ABB RobotStudio station: proyectoRueda.rspag

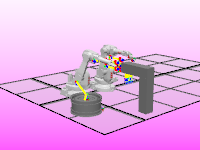
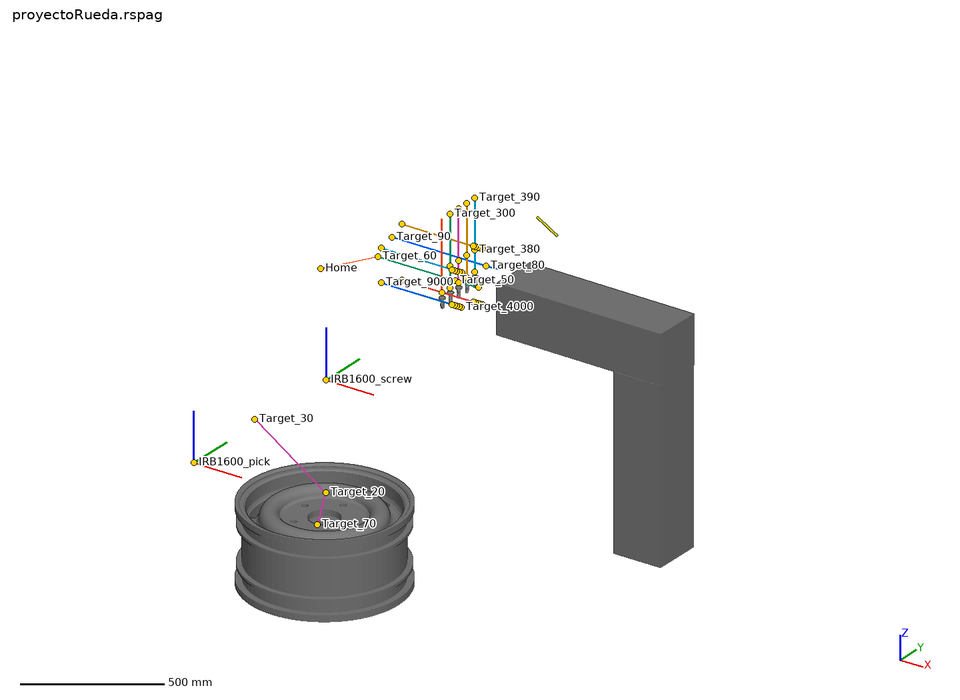
[picture v1: parts stored in the station drawn from their meshes, with robot base, taught points and paths (robot models come from the ABB library and are not in the file)]
--- station ---
Station Versión2 (saved by RobotStudio 21.2.9526.0)
Controller Controlador3, task T_ROB1: task frame (RAPID world) sits at (0, 800, 0) mm in the station
Controller Controlador1
  mechanical unit ROB_1: IRB1600_pick, 6 joints, base frame (0, 0, 0) mm
Controller Controlador3
  mechanical unit ROB_1: IRB1600_screw, 6 joints, base frame (0, 0, 0) mm
Layout (positions relative to the parent item):
  - Pieza_8 [part] at (1800, 250, 0) mm, size 200 x 200 x 700 mm
  - base_rueda [part] at (1800, 450, 700) mm, rotated rx 0 ry 0 rz -0.44 deg, size 700 x 200 x 200 mm
  - IRB1600_pick [mechanism, from Robots\IRB1600_6_120_G_02.rslib] at (0, 0, 0) mm; joint values [0.4149, 0.36, -0.1352, -2.0394, 0.4688, 2.0869] (rad or m)
  - Mi_Ventosa [smart component, from Downloads\1217c23c-7d3e-48fb-b7d3-d1b2005a3c2bMi_Ventosa.rslib] at (890.68, 363.73, 797.26) mm, rotated rx 0 ry 90 rz 0 deg
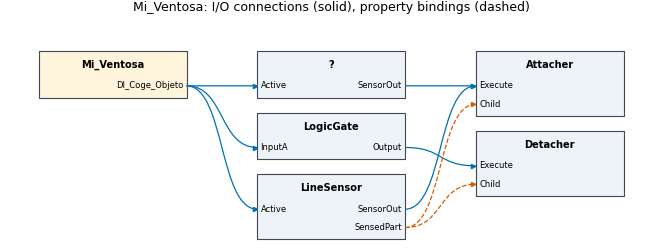
      connections:
        Mi_Ventosa.DI_Coge_Objeto -> ?.Active
        ?.SensorOut -> Attacher.Execute
        Mi_Ventosa.DI_Coge_Objeto -> LogicGate.InputA
        LogicGate.Output -> Detacher.Execute
        Mi_Ventosa.DI_Coge_Objeto -> LineSensor.Active
        LineSensor.SensorOut -> Attacher.Execute
        LineSensor.SensedPart => Attacher.Child
        LineSensor.SensedPart => Detacher.Child
    - Attacher [smart component, from Components\Attacher.rslib]
        properties: Parent=Ventosa; Flange=0; Child=(none); Mount=false; Offset=[0 0 0]; Orientation=[0 0 0]
    - Detacher [smart component, from Components\Detacher.rslib]
        properties: Child=(none); KeepPosition=true
    - Ventosa [mechanism, from Downloads\1217c23c-7d3e-48fb-b7d3-d1b2005a3c2bMi_Ventosa.rslib] at (0, 0, 0) mm
    - LogicGate [smart component, from Components\LogicGate.rslib]
        properties: Operator=NOT; Delay=0
    - LineSensor [smart component, from Components\LineSensor.rslib]
        properties: Start=[0 0 0.055]; End=[0 0 0.07]; Radius=0.001; SensedPart=(none); SensedPoint=[0 0 0]
      - _sensorPart_ [part], size 2 x 2 x 15 mm
    - Indicador [part, from Downloads\1217c23c-7d3e-48fb-b7d3-d1b2005a3c2bMi_Ventosa.rslib] at (-4.38, 0, 0) mm
  - IRB1600_screw [mechanism, from Robots\IRB1600_6_120_G_02.rslib] at (0, 800, 0) mm; joint values [0, 0, 0, 0, 0.5236, 0] (rad or m)
  - Rin [smart component]
    - RC Crawler Wheel Rim 1.9inch Only 5mm Wheel Bore [part] at (899.77, -496.03, 145.15) mm, rotated rx -180 ry 0 rz -180 deg, size 624 x 624 x 312 mm
  - Gripper [smart component]
      signals: DI Cerrar
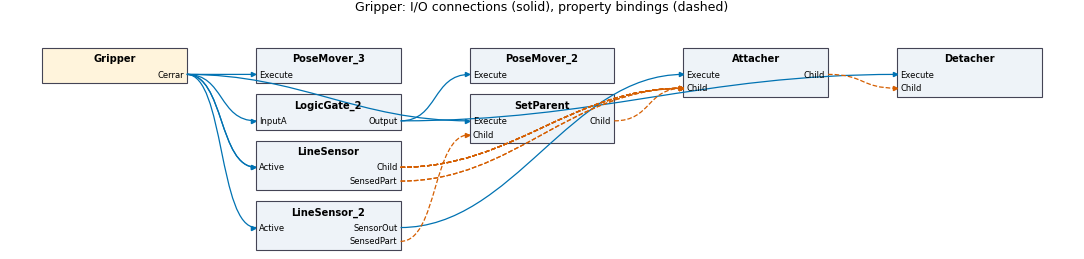
      connections:
        Gripper.Cerrar -> PoseMover_3.Execute
        Gripper.Cerrar -> LogicGate_2.InputA
        LogicGate_2.Output -> PoseMover_2.Execute
        LogicGate_2.Output -> Detacher.Execute
        Gripper.Cerrar -> LineSensor.Active
        Gripper.Cerrar -> VolumeSensor.Active
        Gripper.Cerrar -> LineSensor_2.Active
        Gripper.Cerrar -> SetParent.Execute
        LineSensor_2.SensorOut -> Attacher.Execute
        Attacher.Child => Detacher.Child
        SetParent.Child => Attacher.Child
        SetParent_2.Child => Attacher.Child
        SetParent_3.Child => Attacher.Child
        SetParent_4.Child => Attacher.Child
        SetParent_5.Child => Attacher.Child
        GetParent.Child => Attacher.Child
        LineSensor.SensedPart => Attacher.Child
        VolumeSensor.SensedPart => Attacher.Child
        LineSensor_2.SensedPart => SetParent.Child
        SetParent.Child => Attacher.Child
    - Smart_Gripper_screw [mechanism, from Tools\ABB_Smart_Gripper_Servo_Fingers.rslib] at (806.29, 800, 929) mm, rotated rx 180 ry 60 rz 180 deg; joint values [0.014] (rad or m)
    - PoseMover_2 [smart component, from Components\PoseMover.rslib]
        properties: Mechanism=Smart_Gripper_screw; Pose=2; Duration=1
    - PoseMover_3 [smart component, from Components\PoseMover.rslib]
        properties: Mechanism=Smart_Gripper_screw; Pose=3; Duration=1
    - LogicGate_2 [smart component, from Components\LogicGate.rslib]
        properties: Operator=NOT; Delay=0
    - Attacher [smart component, from Components\Attacher.rslib]
        properties: Parent=Smart_Gripper_screw; Flange=0; Child=(none); Mount=false; Offset=[0 0 0]; Orientation=[0 0 0]
    - Detacher [smart component, from Components\Detacher.rslib]
        properties: Child=(none); KeepPosition=true
    - Indicador [part, from Downloads\1217c23c-7d3e-48fb-b7d3-d1b2005a3c2bMi_Ventosa.rslib] at (-4.38, 0, 0) mm
    - LineSensor_2 [smart component, from Components\LineSensor.rslib] at (891.67, 800, 879.7) mm, rotated rx 180 ry 60 rz 180 deg
        properties: Start=[0 0 0]; End=[0 0 0.1]; Radius=0.004; SensedPart=(none); SensedPoint=[0 0 0]
      - _sensorPart_ [part], size 8 x 8 x 100 mm
    - SetParent [smart component, from Components\SetParent.rslib]
        properties: Child=(none); Parent=(none); KeepTransform=true
  - tornillo2 [smart component] at (0, 3050, 45) mm, rotated rx 0 ry 90 rz 0 deg
    - Pan Cross-head Screw [part] at (0, -1500, 0) mm, size 45.5 x 24 x 24 mm
    - Positioner [smart component, from Components\Positioner.rslib]
        properties: Object=tornillo2; Position=[0 0 0]; Orientation=[0 0 0]; Reference=Global; ReferenceObject=(none)
    - tornillo2_2 [smart component] at (0, 3050, 45) mm, rotated rx 0 ry 90 rz 0 deg
      - Pan Cross-head Screw [part] at (0, -1500, 0) mm, size 45.5 x 24 x 24 mm
      - Positioner [smart component, from Components\Positioner.rslib]
          properties: Object=tornillo2_2; Position=[0 0 0]; Orientation=[0 0 0]; Reference=Global; ReferenceObject=(none)
  - tornillo3 [smart component] at (0, 3100, 45) mm, rotated rx 0 ry 90 rz 0 deg
    - Pan Cross-head Screw [part] at (0, -1500, 0) mm, size 45.5 x 24 x 24 mm
    - Positioner [smart component, from Components\Positioner.rslib]
        properties: Object=tornillo3; Position=[0 0 0]; Orientation=[0 0 0]; Reference=Global; ReferenceObject=(none)
  - tornillo4 [smart component] at (0, 3150, 45) mm, rotated rx 0 ry 90 rz 0 deg
    - Pan Cross-head Screw [part] at (0, -1500, 0) mm, size 45.5 x 24 x 24 mm
    - Positioner [smart component, from Components\Positioner.rslib]
        properties: Object=tornillo4; Position=[0 0 0]; Orientation=[0 0 0]; Reference=Global; ReferenceObject=(none)
  - tornillo5 [smart component] at (0, 3200, 45) mm, rotated rx 0 ry 90 rz 0 deg
    - Pan Cross-head Screw [part] at (0, -1500, 0) mm, size 45.5 x 24 x 24 mm
    - Positioner [smart component, from Components\Positioner.rslib]
        properties: Object=tornillo5; Position=[0 0 0]; Orientation=[0 0 0]; Reference=Global; ReferenceObject=(none)
  - tornillo1.1 [smart component] at (0, 3000, 45) mm, rotated rx 0 ry 90 rz 0 deg
    - Pan Cross-head Screw [part] at (0, -1500, 0) mm, size 45.5 x 24 x 24 mm
    - Positioner [smart component, from Components\Positioner.rslib]
        properties: Object=tornillo1.1; Position=[0 0 0]; Orientation=[0 0 0]; Reference=Global; ReferenceObject=(none)
    - tornillo2_2 [smart component] at (0, 3050, 45) mm, rotated rx 0 ry 90 rz 0 deg
      - Pan Cross-head Screw [part] at (0, -1500, 0) mm, size 45.5 x 24 x 24 mm
      - Positioner [smart component, from Components\Positioner.rslib]
          properties: Object=tornillo2_2; Position=[0 0 0]; Orientation=[0 0 0]; Reference=Global; ReferenceObject=(none)
Attachment: Mi_Ventosa is attached to IRB1600_pick / Link6
Attachment: Smart_Gripper_screw is attached to IRB1600_screw / Link6
Attachment: LineSensor_2 is attached to IRB1600_screw / Link6
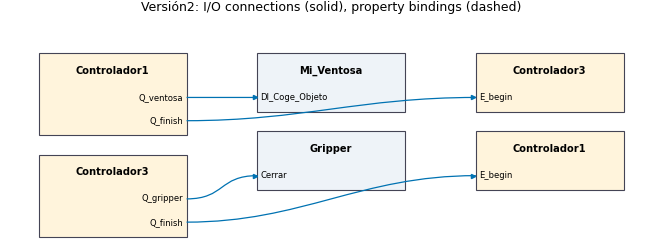
Station logic (signal -> signal, property => property):
  Controlador1.Q_ventosa -> Mi_Ventosa.DI_Coge_Objeto
  Controlador3.Q_gripper -> Gripper.Cerrar
  Controlador3.Q_finish -> Controlador1.E_begin
  Controlador1.Q_finish -> Controlador3.E_begin

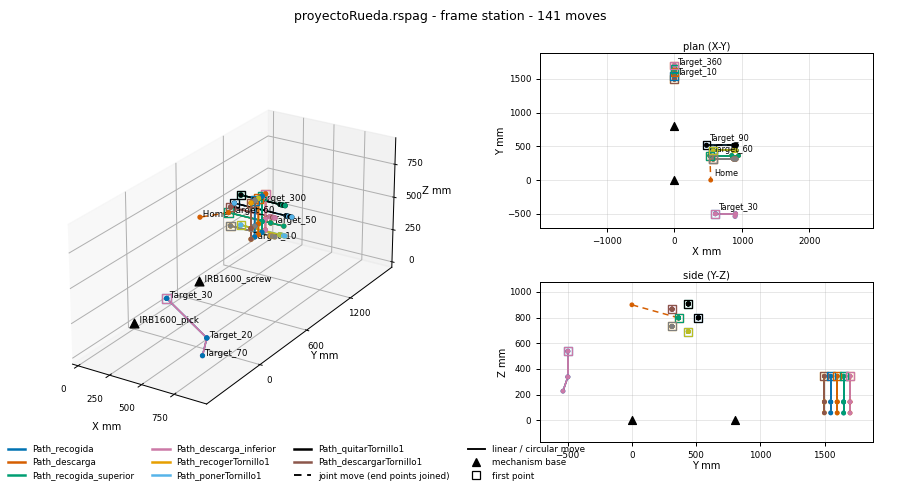
[picture p0: tool path of proyectoRueda.rspag in frame station, 141 of 141 moves have a stored position in this frame; points joined in program order, loops and branches not executed]
--- Backups/Controlador1/RAPID/TASK1/PROGMOD/CalibData.mod ---
MODULE CalibData
    PERS tooldata TCP_Ventosa:=[TRUE,[[0,0,60],[1,0,0,0]],[0.1,[0,0,1],[1,0,0,0],0,0,0]];
    TASK PERS wobjdata WO_recoger:=[FALSE,TRUE,"",[[906.607,-498.004,237.664],[1,0,0,0]],[[0,0,0],[1,0,0,0]]];
    TASK PERS wobjdata WO_descargar:=[FALSE,TRUE,"",[[1038.626,-225.1,0],[1,0,0,0]],[[0,0,0],[1,0,0,0]]];
ENDMODULE

--- Backups/Controlador1/RAPID/TASK1/PROGMOD/Module1.mod ---
MODULE Module1
        CONST robtarget Target_30:=[[-299.326,-0.582,300.001],[0,0,1,0],[-1,0,-1,0],[9E+09,9E+09,9E+09,9E+09,9E+09,9E+09]];
    CONST robtarget Target_20:=[[0.674,-0.582,100.001],[0,0,1,0],[-1,0,-1,0],[9E+09,9E+09,9E+09,9E+09,9E+09,9E+09]];
    CONST robtarget Target_10:=[[0.674,-0.582,0.001],[0,0,1,0],[0,0,0,0],[9E+09,9E+09,9E+09,9E+09,9E+09,9E+09]];
    CONST robtarget Target_60:=[[-512.95,588.826,797.258],[0.707106781,0,0.707106781,0],[0,-2,1,0],[9E+09,9E+09,9E+09,9E+09,9E+09,9E+09]];
    CONST robtarget Target_50:=[[-187.95,588.826,797.258],[0.707106781,0,0.707106781,0],[0,-2,1,0],[9E+09,9E+09,9E+09,9E+09,9E+09,9E+09]];
    CONST robtarget Target_40:=[[-87.95,588.826,797.258],[0.707106781,0,0.707106781,0],[0,-2,1,0],[9E+09,9E+09,9E+09,9E+09,9E+09,9E+09]];
    CONST robtarget Target_70:=[[-7.923,-38.701,-10.664],[0,0,1,0],[-1,0,-1,0],[9E+09,9E+09,9E+09,9E+09,9E+09,9E+09]];
    CONST robtarget Home:=[[-500.958364669,225.1,899],[0.5,0,0.866025404,0],[2,2,-1,6],[9E+09,9E+09,9E+09,9E+09,9E+09,9E+09]];
!***********************************************************
    !
    ! Módulo:  Module1
    !
    ! Descripción:
    !   <Introduzca la descripción aquí>
    !
    ! Autor: KTCHIA
    !
    ! Versión: 1.0
    !
    !***********************************************************


    !***********************************************************
    !
    ! Procedimiento Main
    !
    !   Este es el punto de entrada de su programa
    !
    !***********************************************************
    PROC main()
        !Añada aquí su código
        SetDO Q_finish,0;
        Path_recogida;
        Path_descarga;
        SetDO Q_finish,1;
        WaitDI E_begin,1;
        IF E_begin=1 THEN
            Path_recogida_superior;
            Path_descarga_inferior;
        ENDIF
    ENDPROC
    PROC Path_recogida()
        MoveJ Target_30,v500,z0,TCP_Ventosa\WObj:=WO_recoger;
        MoveL Target_20,v500,z0,TCP_Ventosa\WObj:=WO_recoger;
        MoveL Target_70,v500,z0,TCP_Ventosa\WObj:=WO_recoger;
        SetDO Q_ventosa,1;
        WaitTime 1;
        MoveL Target_20,v500,z0,TCP_Ventosa\WObj:=WO_recoger;
        MoveL Target_30,v500,z0,TCP_Ventosa\WObj:=WO_recoger;
    ENDPROC
    PROC Path_descarga()
        MoveJ Target_60,v500,z0,TCP_Ventosa\WObj:=WO_descargar;
        MoveL Target_50,v500,z0,TCP_Ventosa\WObj:=WO_descargar;
        MoveL Target_40,v500,z0,TCP_Ventosa\WObj:=WO_descargar;
        WaitTime 1;
        MoveL Target_50,v500,z0,TCP_Ventosa\WObj:=WO_descargar;
        SetDO Q_ventosa,0;
        MoveL Target_60,v500,z0,TCP_Ventosa\WObj:=WO_descargar;
        MoveJ Home,v1000,z100,TCP_Ventosa\WObj:=WO_descargar;
    ENDPROC
    PROC Path_recogida_superior()
        MoveJ Target_60,v500,z0,TCP_Ventosa\WObj:=WO_descargar;
        MoveL Target_50,v500,z0,TCP_Ventosa\WObj:=WO_descargar;
        MoveL Target_40,v500,z0,TCP_Ventosa\WObj:=WO_descargar;
        SetDO Q_ventosa,1;
        WaitTime 1;
        MoveL Target_50,v500,z0,TCP_Ventosa\WObj:=WO_descargar;
        MoveL Target_60,v500,z0,TCP_Ventosa\WObj:=WO_descargar;
    ENDPROC
    PROC Path_descarga_inferior()
        MoveJ Target_30,v500,z0,TCP_Ventosa\WObj:=WO_recoger;
        MoveL Target_20,v500,z0,TCP_Ventosa\WObj:=WO_recoger;
        MoveL Target_70,v500,z0,TCP_Ventosa\WObj:=WO_recoger;
        WaitTime 1;
        MoveL Target_20,v500,z0,TCP_Ventosa\WObj:=WO_recoger;
        SetDO Q_ventosa,0;
        MoveL Target_30,v500,z0,TCP_Ventosa\WObj:=WO_recoger;
    ENDPROC
ENDMODULE

--- Backups/Controlador3/RAPID/TASK1/PROGMOD/CalibData.mod ---
MODULE CalibData
    PERS tooldata Servo:=[TRUE,[[0,0,114.2],[1,0,0,0]],[0.215,[8.7,12.3,49.2],[1,0,0,0],0.00021,0.00024,0.00009]];
    TASK PERS wobjdata WO_cogerTornillo:=[FALSE,TRUE,"",[[0,0,0],[1,0,0,0]],[[0,0,0],[1,0,0,0]]];
    TASK PERS wobjdata WO_ponerTornillo:=[FALSE,TRUE,"",[[0,0,0],[1,0,0,0]],[[0,0,0],[1,0,0,0]]];
    TASK PERS wobjdata WO_cogerTornillo1:=[FALSE,TRUE,"",[[0,0,0],[1,0,0,0]],[[0,0,0],[1,0,0,0]]];
    TASK PERS wobjdata WO_ponerTornillo1:=[FALSE,TRUE,"",[[0,0,0],[1,0,0,0]],[[0,0,0],[1,0,0,0]]];
    TASK PERS wobjdata WO_cogerTornillo2:=[FALSE,TRUE,"",[[0,0,0],[1,0,0,0]],[[0,0,0],[1,0,0,0]]];
    TASK PERS wobjdata WO_cogerTornillo3:=[FALSE,TRUE,"",[[0,0,0],[1,0,0,0]],[[0,0,0],[1,0,0,0]]];
    TASK PERS wobjdata WO_cogerTornillo4:=[FALSE,TRUE,"",[[0,0,0],[1,0,0,0]],[[0,0,0],[1,0,0,0]]];
    TASK PERS wobjdata WO_cogerTornillo5:=[FALSE,TRUE,"",[[0,0,0],[1,0,0,0]],[[0,0,0],[1,0,0,0]]];
    TASK PERS wobjdata WO_ponerTornillo2:=[FALSE,TRUE,"",[[0,0,0],[1,0,0,0]],[[0,0,0],[1,0,0,0]]];
    TASK PERS wobjdata WO_ponerTornillo3:=[FALSE,TRUE,"",[[0,0,0],[1,0,0,0]],[[0,0,0],[1,0,0,0]]];
    TASK PERS wobjdata WO_ponerTornillo4:=[FALSE,TRUE,"",[[0,0,0],[1,0,0,0]],[[0,0,0],[1,0,0,0]]];
    TASK PERS wobjdata WO_ponerTornillo5:=[FALSE,TRUE,"",[[0,0,0],[1,0,0,0]],[[0,0,0],[1,0,0,0]]];
ENDMODULE

--- Backups/Controlador3/RAPID/TASK1/PROGMOD/Module1.mod ---
MODULE Module1
        CONST robtarget Target_30:=[[-0.058,698.771,342.903],[0,0,1,0],[1,0,1,0],[9E+09,9E+09,9E+09,9E+09,9E+09,9E+09]];
    CONST robtarget Target_20:=[[-0.058,698.771,142.903],[0,0,1,0],[1,0,1,0],[9E+09,9E+09,9E+09,9E+09,9E+09,9E+09]];
    CONST robtarget Target_10:=[[-0.058,698.771,57.903],[0,0,1,0],[0,0,0,0],[9E+09,9E+09,9E+09,9E+09,9E+09,9E+09]];
    CONST robtarget Target_40:=[[920,-282.5,798],[0.707106781,0,0.707106781,0],[-1,1,-2,0],[9E+09,9E+09,9E+09,9E+09,9E+09,9E+09]];
    CONST robtarget Target_90:=[[475,-282.5,798],[0,0.707106781,0,0.707106781],[-1,1,0,0],[9E+09,9E+09,9E+09,9E+09,9E+09,9E+09]];
    CONST robtarget Target_80:=[[875,-282.5,798],[0,0.707106781,0,0.707106781],[-1,1,0,0],[9E+09,9E+09,9E+09,9E+09,9E+09,9E+09]];
    CONST robtarget Target_70:=[[885,-282.5,798],[0.27059805,-0.653281482,0.27059805,-0.653281482],[-1,1,1,0],[9E+09,9E+09,9E+09,9E+09,9E+09,9E+09]];
    CONST robtarget Target_60:=[[895,-282.5,798],[0.5,-0.5,0.5,-0.5],[-1,1,1,0],[9E+09,9E+09,9E+09,9E+09,9E+09,9E+09]];
    CONST robtarget Target_50:=[[905,-282.5,798],[0.62578076,-0.329239185,0.62578076,-0.329239185],[-1,1,-2,0],[9E+09,9E+09,9E+09,9E+09,9E+09,9E+09]];
    CONST robtarget Target_40_1:=[[910,-282.5,798],[0.694697338,-0.131892411,0.694697338,-0.131892411],[-1,1,-2,0],[9E+09,9E+09,9E+09,9E+09,9E+09,9E+09]];
    CONST robtarget Target_55:=[[905,-282.5,798],[0.653281482,-0.27059805,0.653281482,-0.27059805],[-1,1,-2,0],[9E+09,9E+09,9E+09,9E+09,9E+09,9E+09]];
    CONST robtarget Target_45:=[[915,-282.5,798],[0.707106781,0,0.707106781,0],[-1,1,-2,0],[9E+09,9E+09,9E+09,9E+09,9E+09,9E+09]];
    CONST robtarget Target_56:=[[900,-282.5,798],[0.587937801,-0.392847479,0.587937801,-0.392847479],[-1,1,1,0],[9E+09,9E+09,9E+09,9E+09,9E+09,9E+09]];
    CONST robtarget Target_300:=[[0.2,748.407,342.618],[0,0,1,0],[0,0,0,0],[9E+09,9E+09,9E+09,9E+09,9E+09,9E+09]];
    CONST robtarget Target_200:=[[0.2,748.407,142.618],[0,0,1,0],[0,0,0,0],[9E+09,9E+09,9E+09,9E+09,9E+09,9E+09]];
    CONST robtarget Target_100:=[[0.2,748.407,57.618],[0,0,1,0],[0,0,0,0],[9E+09,9E+09,9E+09,9E+09,9E+09,9E+09]];
    CONST robtarget Target_330:=[[0.975,798.745,343.167],[0,0,1,0],[0,0,0,0],[9E+09,9E+09,9E+09,9E+09,9E+09,9E+09]];
    CONST robtarget Target_320:=[[0.975,798.745,143.167],[0,0,1,0],[0,0,0,0],[9E+09,9E+09,9E+09,9E+09,9E+09,9E+09]];
    CONST robtarget Target_310:=[[0.975,798.745,57.167],[0,0,1,0],[0,0,0,0],[9E+09,9E+09,9E+09,9E+09,9E+09,9E+09]];
    CONST robtarget Target_360:=[[0.487,848.79,342.715],[0,0,1,0],[0,0,0,0],[9E+09,9E+09,9E+09,9E+09,9E+09,9E+09]];
    CONST robtarget Target_350:=[[0.487,848.79,142.715],[0,0,1,0],[0,0,0,0],[9E+09,9E+09,9E+09,9E+09,9E+09,9E+09]];
    CONST robtarget Target_340:=[[0.487,848.79,56.715],[0,0,1,0],[0,0,0,0],[9E+09,9E+09,9E+09,9E+09,9E+09,9E+09]];
    CONST robtarget Target_390:=[[0.244,898.683,343.055],[0,0,1,0],[0,0,0,0],[9E+09,9E+09,9E+09,9E+09,9E+09,9E+09]];
    CONST robtarget Target_380:=[[0.244,898.683,143.055],[0,0,1,0],[0,0,0,0],[9E+09,9E+09,9E+09,9E+09,9E+09,9E+09]];
    CONST robtarget Target_370:=[[0.244,898.683,57.055],[0,0,1,0],[0,0,0,0],[9E+09,9E+09,9E+09,9E+09,9E+09,9E+09]];
    CONST robtarget Target_900:=[[574.529,-360.533,906.323],[0,0.707106781,0,0.707106781],[0,0,0,0],[9E+09,9E+09,9E+09,9E+09,9E+09,9E+09]];
    CONST robtarget Target_400:=[[914.529,-360.533,906.323],[0.707106781,0,0.707106781,0],[-1,1,-2,0],[9E+09,9E+09,9E+09,9E+09,9E+09,9E+09]];
    CONST robtarget Target_500:=[[904.529,-360.533,906.323],[0.653281482,-0.27059805,0.653281482,-0.27059805],[-1,1,-2,0],[9E+09,9E+09,9E+09,9E+09,9E+09,9E+09]];
    CONST robtarget Target_600:=[[894.529,-360.533,906.323],[0.5,-0.5,0.5,-0.5],[-1,1,1,0],[9E+09,9E+09,9E+09,9E+09,9E+09,9E+09]];
    CONST robtarget Target_700:=[[884.529,-360.533,906.323],[0.27059805,-0.653281482,0.27059805,-0.653281482],[-1,1,1,0],[9E+09,9E+09,9E+09,9E+09,9E+09,9E+09]];
    CONST robtarget Target_800:=[[874.529,-360.533,906.323],[0,0.707106781,0,0.707106781],[-1,1,0,0],[9E+09,9E+09,9E+09,9E+09,9E+09,9E+09]];
    CONST robtarget Target_990:=[[574.529,-487.2,865.271],[0,0.707106781,0,0.707106781],[0,0,0,0],[9E+09,9E+09,9E+09,9E+09,9E+09,9E+09]];
    CONST robtarget Target_940:=[[914.529,-487.2,865.271],[0.707106781,0,0.707106781,0],[-1,1,-2,0],[9E+09,9E+09,9E+09,9E+09,9E+09,9E+09]];
    CONST robtarget Target_950:=[[904.529,-487.2,865.271],[0.653281482,-0.27059805,0.653281482,-0.27059805],[-1,1,-2,0],[9E+09,9E+09,9E+09,9E+09,9E+09,9E+09]];
    CONST robtarget Target_960:=[[894.529,-487.2,865.271],[0.5,-0.5,0.5,-0.5],[-1,1,1,0],[9E+09,9E+09,9E+09,9E+09,9E+09,9E+09]];
    CONST robtarget Target_970:=[[884.529,-487.2,865.271],[0.27059805,-0.653281482,0.27059805,-0.653281482],[-1,1,1,0],[9E+09,9E+09,9E+09,9E+09,9E+09,9E+09]];
    CONST robtarget Target_980:=[[874.529,-487.2,865.271],[0,0.707106781,0,0.707106781],[-1,1,0,0],[9E+09,9E+09,9E+09,9E+09,9E+09,9E+09]];
    CONST robtarget Target_9000:=[[574.029,-487.592,731.451],[0,0.707106781,0,0.707106781],[0,0,0,0],[9E+09,9E+09,9E+09,9E+09,9E+09,9E+09]];
    CONST robtarget Target_4000:=[[914.029,-487.592,731.451],[0.707106781,0,0.707106781,0],[-1,1,-2,0],[9E+09,9E+09,9E+09,9E+09,9E+09,9E+09]];
    CONST robtarget Target_5000:=[[904.029,-487.592,731.451],[0.653281482,-0.27059805,0.653281482,-0.27059805],[-1,1,-2,0],[9E+09,9E+09,9E+09,9E+09,9E+09,9E+09]];
    CONST robtarget Target_6000:=[[894.029,-487.592,731.451],[0.5,-0.5,0.5,-0.5],[-1,1,1,0],[9E+09,9E+09,9E+09,9E+09,9E+09,9E+09]];
    CONST robtarget Target_7000:=[[884.029,-487.592,731.451],[0.27059805,-0.653281482,0.27059805,-0.653281482],[-1,1,1,0],[9E+09,9E+09,9E+09,9E+09,9E+09,9E+09]];
    CONST robtarget Target_8000:=[[874.029,-487.592,731.451],[0,0.707106781,0,0.707106781],[-1,1,0,0],[9E+09,9E+09,9E+09,9E+09,9E+09,9E+09]];
    CONST robtarget Target_9090:=[[574.029,-360.611,690.519],[0,0.707106781,0,0.707106781],[0,0,0,0],[9E+09,9E+09,9E+09,9E+09,9E+09,9E+09]];
    CONST robtarget Target_9040:=[[914.029,-360.611,690.519],[0.707106781,0,0.707106781,0],[-1,1,-2,0],[9E+09,9E+09,9E+09,9E+09,9E+09,9E+09]];
    CONST robtarget Target_9050:=[[904.029,-360.611,690.519],[0.653281482,-0.27059805,0.653281482,-0.27059805],[-1,1,1,0],[9E+09,9E+09,9E+09,9E+09,9E+09,9E+09]];
    CONST robtarget Target_9060:=[[894.029,-360.611,690.519],[0.5,-0.5,0.5,-0.5],[-1,1,1,0],[9E+09,9E+09,9E+09,9E+09,9E+09,9E+09]];
    CONST robtarget Target_9070:=[[884.029,-360.611,690.519],[0.27059805,-0.653281482,0.27059805,-0.653281482],[-1,1,0,0],[9E+09,9E+09,9E+09,9E+09,9E+09,9E+09]];
    CONST robtarget Target_9080:=[[874.029,-360.611,690.519],[0,0.707106781,0,0.707106781],[-1,1,0,0],[9E+09,9E+09,9E+09,9E+09,9E+09,9E+09]];
!***********************************************************
    !
    ! Módulo:  Module1
    !
    ! Descripción:
    !   <Introduzca la descripción aquí>
    !
    ! Autor: KTCHIA
    !
    ! Versión: 1.0
    !
    !***********************************************************


    !***********************************************************
    !
    ! Procedimiento Main
    !
    !   Este es el punto de entrada de su programa
    !
    !***********************************************************
    PROC main()
        !Añada aquí su código}
        SetDO Q_finish,0;
        IF E_begin=0 THEN
            WaitDI E_begin,1;
        ENDIF
        IF E_begin = 1 THEN
            SetDO Q_gripper,0;
            Path_recogerTornillo1;
            Path_ponerTornillo1;
            Path_recogerTornillo2;
            Path_ponerTornillo2;
            Path_recogerTornillo3;
            Path_ponerTornillo3;
            Path_recogerTornillo4;
            Path_ponerTornillo4;
            Path_recogerTornillo5;
            Path_ponerTornillo5;
            Path_quitarTornillo1;
            Path_descargarTornillo1;
            Path_quitarTornillo2;
            Path_descargarTornillo2;
            Path_quitarTornillo3;
            Path_descargarTornillo3;
            Path_quitarTornillo4;
            Path_descargarTornillo4;
            Path_quitarTornillo5;
            Path_descargarTornillo5;
            SetDO Q_finish,1;
        ENDIF
    ENDPROC

    PROC Path_recogerTornillo1()
        MoveJ Target_30,v500,fine,Servo\WObj:=WO_cogerTornillo1;
        SetDO Q_gripper,0;
        WaitTime 1;
        MoveL Target_20,v500,fine,Servo\WObj:=WO_cogerTornillo1;
        MoveL Target_10,v500,fine,Servo\WObj:=WO_cogerTornillo1;
        SetDO Q_gripper,1;
        WaitTime 1;
        MoveL Target_20,v500,fine,Servo\WObj:=WO_cogerTornillo1;
        MoveL Target_30,v500,fine,Servo\WObj:=WO_cogerTornillo1;
    ENDPROC
    PROC Path_ponerTornillo1()
        MoveJ Target_90,v500,fine,Servo\WObj:=WO_ponerTornillo1;
        MoveL Target_80,v500,fine,Servo\WObj:=WO_ponerTornillo1;
        MoveL Target_70,v500,fine,Servo\WObj:=WO_ponerTornillo1;
        MoveJ Target_60,v500,fine,Servo\WObj:=WO_ponerTornillo1;
        SetDO Q_gripper,0;
        WaitTime 1;
        MoveJ Target_50,v500,fine,Servo\WObj:=WO_ponerTornillo1;
        SetDO Q_gripper,1;
        WaitTime 1;
        MoveJ Target_40,v500,fine,Servo\WObj:=WO_ponerTornillo1;
        SetDO Q_gripper,0;
        WaitTime 1;
        MoveL Target_90,v500,fine,Servo\WObj:=WO_ponerTornillo1;
    ENDPROC
    PROC Path_quitarTornillo1()
        MoveJ Target_90,v500,fine,Servo\WObj:=WO_ponerTornillo1;
        MoveL Target_40,v500,fine,Servo\WObj:=WO_ponerTornillo1;
        SetDO Q_gripper,1;
        WaitTime 1;
        MoveJ Target_50,v500,fine,Servo\WObj:=WO_ponerTornillo1;
        SetDO Q_gripper,0;
        WaitTime 1;
        MoveJ Target_60,v500,fine,Servo\WObj:=WO_ponerTornillo1;
        SetDO Q_gripper,1;
        WaitTime 1;
        MoveL Target_70,v500,fine,Servo\WObj:=WO_ponerTornillo1;
        MoveL Target_80,v500,fine,Servo\WObj:=WO_ponerTornillo1;
        MoveJ Target_90,v500,fine,Servo\WObj:=WO_ponerTornillo1;
    ENDPROC
    PROC Path_descargarTornillo1()
        MoveJ Target_30,v500,fine,Servo\WObj:=WO_cogerTornillo1;
        MoveL Target_20,v500,fine,Servo\WObj:=WO_cogerTornillo1;
        MoveL Target_10,v500,fine,Servo\WObj:=WO_cogerTornillo1;
        SetDO Q_gripper,0;
        WaitTime 1;
        MoveL Target_20,v500,fine,Servo\WObj:=WO_cogerTornillo1;
        MoveL Target_30,v500,fine,Servo\WObj:=WO_cogerTornillo1;
    ENDPROC
    PROC Path_recogerTornillo2()
        SetDO Q_gripper,0;
        MoveJ Target_300,v500,fine,Servo\WObj:=WO_cogerTornillo2;
        WaitTime 1;
        MoveL Target_200,v500,fine,Servo\WObj:=WO_cogerTornillo2;
        MoveL Target_100,v500,fine,Servo\WObj:=WO_cogerTornillo2;
        SetDO Q_gripper,1;
        WaitTime 3;
        MoveL Target_200,v500,fine,Servo\WObj:=WO_cogerTornillo2;
        MoveL Target_300,v500,fine,Servo\WObj:=WO_cogerTornillo2;
    ENDPROC
    PROC Path_recogerTornillo3()
        MoveJ Target_330,v500,fine,Servo\WObj:=WO_cogerTornillo3;
        SetDO Q_gripper,0;
        WaitTime 1;
        MoveL Target_320,v500,fine,Servo\WObj:=WO_cogerTornillo3;
        MoveL Target_310,v500,fine,Servo\WObj:=WO_cogerTornillo3;
        SetDO Q_gripper,1;
        WaitTime 1;
        MoveL Target_320,v500,fine,Servo\WObj:=WO_cogerTornillo3;
        MoveL Target_330,v500,fine,Servo\WObj:=WO_cogerTornillo3;
    ENDPROC
    PROC Path_recogerTornillo4()
        MoveJ Target_360,v500,fine,Servo\WObj:=WO_cogerTornillo4;
        SetDO Q_gripper,0;
        WaitTime 1;
        MoveL Target_350,v500,fine,Servo\WObj:=WO_cogerTornillo4;
        MoveL Target_340,v500,fine,Servo\WObj:=WO_cogerTornillo4;
        SetDO Q_gripper,1;
        WaitTime 1;
        MoveL Target_350,v500,fine,Servo\WObj:=WO_cogerTornillo4;
        MoveL Target_360,v500,fine,Servo\WObj:=WO_cogerTornillo4;
    ENDPROC
    PROC Path_recogerTornillo5()
        MoveJ Target_390,v500,fine,Servo\WObj:=WO_cogerTornillo5;
        SetDO Q_gripper,0;
        WaitTime 1;
        MoveL Target_380,v500,fine,Servo\WObj:=WO_cogerTornillo5;
        MoveL Target_370,v500,fine,Servo\WObj:=WO_cogerTornillo5;
        SetDO Q_gripper,1;
        WaitTime 1;
        MoveL Target_380,v500,fine,Servo\WObj:=WO_cogerTornillo5;
        MoveL Target_390,v500,fine,Servo\WObj:=WO_cogerTornillo5;
    ENDPROC
    PROC Path_quitarTornillo2()
        MoveJ Target_900,v500,fine,Servo\WObj:=WO_ponerTornillo2;
        MoveL Target_400,v500,fine,Servo\WObj:=WO_ponerTornillo2;
        SetDO Q_gripper,1;
        WaitTime 1;
        MoveL Target_500,v500,fine,Servo\WObj:=WO_ponerTornillo2;
        SetDO Q_gripper,0;
        WaitTime 1;
        MoveL Target_600,v500,fine,Servo\WObj:=WO_ponerTornillo2;
        SetDO Q_gripper,1;
        WaitTime 1;
        MoveL Target_700,v500,fine,Servo\WObj:=WO_ponerTornillo2;
        MoveL Target_800,v500,fine,Servo\WObj:=WO_ponerTornillo2;
        MoveL Target_900,v500,fine,Servo\WObj:=WO_ponerTornillo2;
    ENDPROC
    PROC Path_quitarTornillo3()
        MoveJ Target_990,v500,fine,Servo\WObj:=WO_ponerTornillo3;
        MoveL Target_940,v500,fine,Servo\WObj:=WO_ponerTornillo3;
        SetDO Q_gripper,1;
        WaitTime 1;
        MoveL Target_950,v500,fine,Servo\WObj:=WO_ponerTornillo3;
        SetDO Q_gripper,0;
        WaitTime 1;
        MoveL Target_960,v500,fine,Servo\WObj:=WO_ponerTornillo3;
        SetDO Q_gripper,1;
        WaitTime 1;
        MoveL Target_970,v500,fine,Servo\WObj:=WO_ponerTornillo3;
        MoveL Target_980,v500,fine,Servo\WObj:=WO_ponerTornillo3;
        MoveL Target_990,v500,fine,Servo\WObj:=WO_ponerTornillo3;
    ENDPROC
    PROC Path_quitarTornillo4()
        MoveJ Target_9000,v500,fine,Servo\WObj:=WO_ponerTornillo4;
        MoveL Target_4000,v500,fine,Servo\WObj:=WO_ponerTornillo4;
        SetDO Q_gripper,1;
        WaitTime 1;
        MoveL Target_5000,v500,fine,Servo\WObj:=WO_ponerTornillo4;
        SetDO Q_gripper,0;
        WaitTime 1;
        MoveL Target_6000,v500,fine,Servo\WObj:=WO_ponerTornillo4;
        SetDO Q_gripper,1;
        WaitTime 1;
        MoveL Target_7000,v500,fine,Servo\WObj:=WO_ponerTornillo4;
        MoveL Target_8000,v500,fine,Servo\WObj:=WO_ponerTornillo4;
        MoveL Target_9000,v500,fine,Servo\WObj:=WO_ponerTornillo4;
    ENDPROC
    PROC Path_quitarTornillo5()
        MoveJ Target_9090,v500,fine,Servo\WObj:=WO_ponerTornillo5;
        MoveL Target_9040,v500,fine,Servo\WObj:=WO_ponerTornillo5;
        SetDO Q_gripper,1;
        WaitTime 1;
        MoveL Target_9050,v500,fine,Servo\WObj:=WO_ponerTornillo5;
        SetDO Q_gripper,0;
        WaitTime 1;
        MoveL Target_9060,v500,fine,Servo\WObj:=WO_ponerTornillo5;
        SetDO Q_gripper,1;
        WaitTime 1;
        MoveL Target_9070,v500,fine,Servo\WObj:=WO_ponerTornillo5;
        MoveL Target_9080,v500,fine,Servo\WObj:=WO_ponerTornillo5;
        MoveL Target_9090,v500,fine,Servo\WObj:=WO_ponerTornillo5;
    ENDPROC
    PROC Path_ponerTornillo2()
        MoveJ Target_900,v500,fine,Servo\WObj:=WO_ponerTornillo2;
        MoveL Target_800,v500,fine,Servo\WObj:=WO_ponerTornillo2;
        MoveL Target_700,v500,fine,Servo\WObj:=WO_ponerTornillo2;
        MoveL Target_600,v500,fine,Servo\WObj:=WO_ponerTornillo2;
        SetDO Q_gripper,0;
        WaitTime 1;
        MoveL Target_500,v500,fine,Servo\WObj:=WO_ponerTornillo2;
        SetDO Q_gripper,1;
        WaitTime 1;
        MoveL Target_400,v500,fine,Servo\WObj:=WO_ponerTornillo2;
        SetDO Q_gripper,0;
        WaitTime 1;
        MoveL Target_900,v500,fine,Servo\WObj:=WO_ponerTornillo2;
    ENDPROC
    PROC Path_ponerTornillo3()
        MoveJ Target_990,v500,fine,Servo\WObj:=WO_ponerTornillo3;
        MoveL Target_980,v500,fine,Servo\WObj:=WO_ponerTornillo3;
        MoveL Target_970,v500,fine,Servo\WObj:=WO_ponerTornillo3;
        MoveL Target_960,v500,fine,Servo\WObj:=WO_ponerTornillo3;
        SetDO Q_gripper,0;
        WaitTime 1;
        MoveL Target_950,v500,fine,Servo\WObj:=WO_ponerTornillo3;
        SetDO Q_gripper,1;
        WaitTime 1;
        MoveL Target_940,v500,fine,Servo\WObj:=WO_ponerTornillo3;
        SetDO Q_gripper,0;
        WaitTime 1;
        MoveL Target_990,v500,fine,Servo\WObj:=WO_ponerTornillo3;
    ENDPROC
    PROC Path_ponerTornillo4()
        MoveJ Target_9000,v500,fine,Servo\WObj:=WO_ponerTornillo4;
        MoveL Target_8000,v500,fine,Servo\WObj:=WO_ponerTornillo4;
        MoveL Target_7000,v500,fine,Servo\WObj:=WO_ponerTornillo4;
        MoveL Target_6000,v500,fine,Servo\WObj:=WO_ponerTornillo4;
        SetDO Q_gripper,0;
        WaitTime 1;
        MoveL Target_5000,v500,fine,Servo\WObj:=WO_ponerTornillo4;
        SetDO Q_gripper,1;
        WaitTime 1;
        MoveL Target_4000,v500,fine,Servo\WObj:=WO_ponerTornillo4;
        SetDO Q_gripper,0;
        WaitTime 1;
        MoveL Target_9000,v500,fine,Servo\WObj:=WO_ponerTornillo4;
    ENDPROC
    PROC Path_ponerTornillo5()
        MoveJ Target_9090,v500,fine,Servo\WObj:=WO_ponerTornillo5;
        MoveL Target_9080,v500,fine,Servo\WObj:=WO_ponerTornillo5;
        MoveL Target_9070,v500,fine,Servo\WObj:=WO_ponerTornillo5;
        MoveL Target_9060,v500,fine,Servo\WObj:=WO_ponerTornillo5;
        SetDO Q_gripper,0;
        WaitTime 1;
        MoveL Target_9050,v500,fine,Servo\WObj:=WO_ponerTornillo5;
        SetDO Q_gripper,1;
        WaitTime 1;
        MoveL Target_9040,v500,fine,Servo\WObj:=WO_ponerTornillo5;
        SetDO Q_gripper,0;
        WaitTime 1;
        MoveL Target_9090,v500,fine,Servo\WObj:=WO_ponerTornillo5;
    ENDPROC
    PROC Path_descargarTornillo2()
        MoveJ Target_300,v500,fine,Servo\WObj:=WO_cogerTornillo2;
        MoveL Target_200,v500,fine,Servo\WObj:=WO_cogerTornillo2;
        MoveL Target_100,v500,fine,Servo\WObj:=WO_cogerTornillo2;
        SetDO Q_gripper,0;
        WaitTime 1;
        MoveL Target_200,v500,fine,Servo\WObj:=WO_cogerTornillo2;
        MoveL Target_300,v500,fine,Servo\WObj:=WO_cogerTornillo2;
    ENDPROC
    PROC Path_descargarTornillo3()
        MoveJ Target_330,v500,fine,Servo\WObj:=WO_cogerTornillo3;
        MoveL Target_320,v500,fine,Servo\WObj:=WO_cogerTornillo3;
        MoveL Target_310,v500,fine,Servo\WObj:=WO_cogerTornillo3;
        SetDO Q_gripper,0;
        WaitTime 1;
        MoveL Target_320,v500,fine,Servo\WObj:=WO_cogerTornillo3;
        MoveL Target_330,v500,fine,Servo\WObj:=WO_cogerTornillo3;
    ENDPROC
    PROC Path_descargarTornillo4()
        MoveJ Target_360,v500,fine,Servo\WObj:=WO_cogerTornillo4;
        MoveL Target_350,v500,fine,Servo\WObj:=WO_cogerTornillo4;
        MoveL Target_340,v500,fine,Servo\WObj:=WO_cogerTornillo4;
        SetDO Q_gripper,0;
        WaitTime 1;
        MoveL Target_350,v500,fine,Servo\WObj:=WO_cogerTornillo4;
        MoveL Target_360,v500,fine,Servo\WObj:=WO_cogerTornillo4;
    ENDPROC
    PROC Path_descargarTornillo5()
        MoveJ Target_390,v500,fine,Servo\WObj:=WO_cogerTornillo5;
        MoveL Target_380,v500,fine,Servo\WObj:=WO_cogerTornillo5;
        MoveL Target_370,v500,fine,Servo\WObj:=WO_cogerTornillo5;
        SetDO Q_gripper,0;
        WaitTime 1;
        MoveL Target_380,v500,fine,Servo\WObj:=WO_cogerTornillo5;
        MoveL Target_390,v500,fine,Servo\WObj:=WO_cogerTornillo5;
    ENDPROC
ENDMODULE

--- Backups/Controlador1/SYSPAR/EIO.cfg ---
EIO:CFG_1.0:6:1::
#
EIO_SIGNAL:

      -Name "Q_ventosa" -SignalType "DO"

      -Name "Q_finish" -SignalType "DO"

      -Name "E_begin" -SignalType "DI"

--- Backups/Controlador3/SYSPAR/EIO.cfg ---
EIO:CFG_1.0:6:1::
#
EIO_SIGNAL:

      -Name "Q_gripper" -SignalType "DO"

      -Name "Q_finish" -SignalType "DO"

      -Name "E_begin" -SignalType "DI"
